FUNCTION_BLOCK SelectMode (* Basic Function Block Type *)
  (* Standard: 61499-2 *)
  (* Version 0.0, 3/27/2024, SESA371406, Schneider Electric, Template *)
  PACKAGE SE.Nereda;
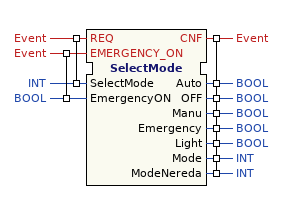
  EVENT_INPUT
    REQ WITH SelectMode; (* Normal Execution Request *)
    EMERGENCY_ON WITH EmergencyON;
  END_EVENT
  EVENT_OUTPUT
    CNF WITH Auto, OFF, Manu, Emergency, Light, Mode, ModeNereda; (* Execution Confirmation *)
  END_EVENT
  VAR_INPUT
    SelectMode : INT;
    EmergencyON : BOOL;
  END_VAR
  VAR_OUTPUT
    Auto : BOOL;
    OFF : BOOL;
    Manu : BOOL;
    Emergency : BOOL;
    Light : BOOL;
    Mode : INT;
    ModeNereda : INT;
  END_VAR
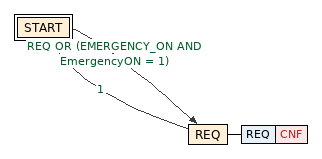
  EC_STATES
    START; (* Initial State *)
    REQ : REQ -> CNF; (* Normal execution *)
  END_STATES
  EC_TRANSITIONS
    START TO REQ := REQ OR (EMERGENCY_ON AND EmergencyON = 1);
    REQ TO START := 1;
  END_TRANSITIONS
  ALGORITHM REQ IN ST: (* Normally executed algorithm *)
;
IF SelectMode = 0 AND EmergencyON = FALSE THEN // Auto mode selected and communication is healthy
	// Activate Auto mode
	Auto := TRUE;
	OFF := FALSE;
	Manu := FALSE;
	Emergency := FALSE;

	// Turn ON mode indication light
	Light := TRUE;

	// Set current mode value to Auto
	Mode := 0;
	ModeNereda:=2;

ELSIF SelectMode = 1 THEN // OFF mode selected

	// Activate OFF mode
	Auto := FALSE;
	OFF := TRUE;
	Manu := FALSE;
	Emergency := FALSE;

	// Turn OFF mode indication light
	Light := FALSE;

	// Set current mode value to OFF
	Mode := 1;
	ModeNereda:=0;

ELSIF SelectMode = 2 THEN // Manual mode selected

	// Activate Manual mode
	Auto := FALSE;
	OFF := FALSE;
	Manu := TRUE;
	Emergency := FALSE;

	// Turn ON mode indication light
	Light := TRUE;

	// Set current mode value to Manual
	Mode := 2;
	ModeNereda:=1;

ELSIF SelectMode = 3 OR (EmergencyON = TRUE AND SelectMode = 0) THEN // Emergency mode selected or Auto mode with communication failure

	// Activate Emergency mode
	Auto := FALSE;
	OFF := FALSE;
	Manu := FALSE;
	Emergency := TRUE;

	// Turn ON mode indication light
	Light := TRUE;

	// Set current mode value to Emergency
	Mode := 3;
	ModeNereda:=-1;

END_IF;
  END_ALGORITHM
END_FUNCTION_BLOCK
